TYPE ST_ValveCommand :
STRUCT
	bMove        : BOOL;
    bStop        : BOOL;
    iTargetPos   : INT; // 1..6
    bBusy        : BOOL;
END_STRUCT
END_TYPE

(* stored: Version 1.1.0.1, ProductVersion 3.1.4024.12
   DUT ST_ValveCommand: Id {c73469e4-e9ca-4d95-bd9d-3015d4dd47d6} *)
